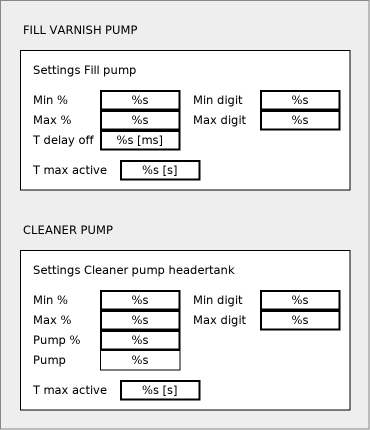
VISUALIZATION VISU_SETTINGS  // 370x430
    Rectangle (0,0 370x430)
    Rectangle (20,20 250x20), "FILL VARNISH PUMP"
    Rectangle (20,50 330x140)
    Rectangle (30,90 70x20), "Min %"
    Rectangle (30,110 70x20), "Max %"
    Rectangle (30,60 260x20), "Settings Fill pump"
    Rectangle (100,90 80x20), "%s", text variable: PRG_INK.wIDp_MinSpeedFillInkPumpVarnish
        OnMouseDown: write the text variable via Edit, min 0, max 100
    Rectangle (100,110 80x20), "%s", text variable: PRG_INK.wIDp_MaxSpeedFillInkPumpVarnish
        OnMouseDown: write the text variable via Edit, min 0, max 100
    Rectangle (100,130 80x20), "%s [ms]", text variable: PRG_INK.wIDp_PumpTimeOffDelayVarnish
        OnMouseDown: write the text variable via Edit
    Rectangle (30,130 70x20), "T delay off"
    Rectangle (190,90 70x20), "Min digit"
    Rectangle (190,110 70x20), "Max digit"
    Rectangle (260,90 80x20), "%s", text variable: PRG_INK.wIDP_AnalogMinDigitVarnish
        OnMouseDown: write the text variable via Edit, min 0, max 65535
    Rectangle (260,110 80x20), "%s", text variable: PRG_INK.wIDP_AnalogMaxDigitVarnish
        OnMouseDown: write the text variable via Edit, min 0, max 65535
    Rectangle (30,160 86x20), "T max active"
    Rectangle (120,160 80x20), "%s [s]", text variable: PRG_INK.sC_Config_I.wC_INKPUMP_MAX_TIME
        OnMouseDown: write the text variable via Edit
    Rectangle (20,220 250x20), "CLEANER PUMP"
    Rectangle (20,250 330x160)
    Rectangle (30,260 250x20), "Settings Cleaner pump headertank"
    Rectangle (30,290 70x20), "Min %"
    Rectangle (30,310 70x20), "Max %"
    Rectangle (30,350 70x20), "Pump"
    Rectangle (100,290 80x20), "%s", text variable: PRG_INK.lR_MinSpeedFillInkPumpCleaner
        OnMouseDown: write the text variable via Edit
    Rectangle (100,310 80x20), "%s", text variable: PRG_INK.lR_MaxSpeedFillInkPumpCleaner
        OnMouseDown: write the text variable via Edit
    Rectangle (100,350 80x20), "%s", text variable: PRG_INK.wL_StptSpeedCleanInkPumpDigit
    Rectangle (100,330 80x20), "%s", text variable: PRG_INK.lR_StptSpeedCleanInkPumpCleanerPercent
        OnMouseDown: write the text variable via Edit
    Rectangle (30,330 70x20), "Pump %"
    Rectangle (190,290 70x20), "Min digit"
    Rectangle (190,310 70x20), "Max digit"
    Rectangle (260,290 80x20), "%s", text variable: PRG_INK.lR_AnalogMinDigitCleaner
        OnMouseDown: write the text variable via Edit, min 0, max 65535
    Rectangle (260,310 80x20), "%s", text variable: PRG_INK.lR_AnalogMaxDigitCleaner
        OnMouseDown: write the text variable via Edit, min 0, max 65535
    Rectangle (30,380 86x20), "T max active"
    Rectangle (120,380 80x20), "%s [s]", text variable: PRG_INK.sC_Config_I.wC_CLEANERPUMP_MAX_TIME
        OnMouseDown: write the text variable via Edit
END_VISUALIZATION

(* stored: Version 1.1.0.1, ProductVersion 3.1.4024.3
   Visu VISU_SETTINGS: Id {0ef5a966-9586-445b-b8d7-b949545be274} *)
